Staubli VAL3: createLicense.pgx

program createLicense()
  local string txt[6]
  local string orderNumber
  local num i
 begin
    //\brief
  // Create a license key for the robot system. License key information is saved
  // in system data library
  //
  //\var txt
  //\var orderNumber
  //\var i
  //
//!brief
  // Create a license key for the robot system. License key information is saved
  // in system data library
  //
  orderNumber=getVersion("serialNumber")
  txt=""
  //!issue 36
  if data:libLoad("zData")==0
    call list:resizeNum(data:nLic,len(orderNumber))
    data:sMachineNumber=orderNumber
    for i=0 to size(data:nLic)-1
      data:nLic[i]=asc(orderNumber,i)*(i+1)
      txt=txt+toString("",asc(orderNumber,i)*(i+1))+", "
    endFor
    call data:saveData()
    popUpMsg(txt)
  else
    popUpMsg("Loading the data library failed!")
  endIf
end
